(* Logix 5000 project; controller QA_DC vendor 1 type 14 code 164 rev 32.16; software revision 32.04; part 2 of 3 *)
(* tags used below, declared in another part *)
   LN98_1st_Station_Break_Code : DINT;
   LN98_Break_LineWide : BOOL;
   LN98_FROM_DC1_MAIN_MESSAGES : DINT[20];
   LN98_Schedule : UDT_Current_Status;
   LN98_TO_DC1_MAIN_MESSAGE_E : DINT[10];   // WORK CENTER E CONSUME TAG
   LN98_TO_DC1_SUB_MESSAGE_E : DINT[10];   // WORK CENTER E CONSUME TAG
   LN98EES01 : DINT;
   LN98EES02 : DINT;
   LN98EES03 : DINT;
   LN98NEM02 : DINT;
   LN98NEM03 : DINT;
   LN98NEM04 : DINT;
   LN98NEM05 : DINT;
   LN98SEM02 : DINT;
   LN98SEM04 : DINT;
   LN98SEM05 : DINT;
   LN98WES01 : DINT;
   LN98WES02 : DINT;
   LN98WES03 : DINT;
   LN99_1st_Station_Break_Code : DINT;
   LN99_Break_LineWide : BOOL;
   LN99_Current_Shift_Duration_Mins : DINT;
   LN99_Current_Shift_Duration_wBreaks_Mins : DINT;
   LN99_DC_Controlled_Theoretical_Units : BOOL;
   LN99_DT_CODE : DINT;
   LN99_NewDataModelSerial : BOOL;
   LN99_PreviousSerialNumber : STRING;
   LN99_Schedule : UDT_Current_Status;
   LN99_Schedule_Cycle_Timer : TIMER;
   LN99_Schedule_Max_Break_Duration : DINT;
   LN99_Schedule_Max_Break_Timer : TIMER;
   LN99_Schedule_TAKT : REAL;
   LN99_Scheduled_Units_Buffer : DINT;
   LN99_SerialNumber_ONS : BOOL;
   LN99_SerialNumberBuffer : STRING;
   LN99_SerialNumberChange_DelayTimer : TIMER;
   LN99_SerialNumberChange_Timer : TIMER;
   LN99_Shift_Reset_ONS : BOOL;
   LN99_Theoretical_Units_Counter : COUNTER;
   LN99_Theoretical_Units_Counter_ONS : BOOL;
   LN99_TO_DC01_DOWNTIME_CODE : DINT[10];   // DOWNTIME CODE CONSUME TAG
   LN99_TO_DC01_MAIN_MESSAGES : DINT[20];   // KPI CONSUME TAG
   LN99_TO_DC01_MODEL_SERIAL_MESSAGE : STRING[2];
   LN99_TO_DC1_MAIN_MESSAGE_A : DINT[10];   // WORK CENTER A CONSUME TAG
   LN99_TO_DC1_MAIN_MESSAGE_B : DINT[10];   // WORK CENTER B CONSUME TAG
   LN99_TO_DC1_MAIN_MESSAGE_C : DINT[10];   // WORK CENTER C CONSUME TAG
   LN99_Weekly_Schedule : UDT_Weekly_Schedule;
   LN99_WORKCENTER_MAINLINE_A_DT_CODE : DINT;
   LN99_WORKCENTER_MAINLINE_B_DT_CODE : DINT;
   LN99_WORKCENTER_MAINLINE_C_DT_CODE : DINT;
   LN99_WORKCENTER_MAINLINE_D_DT_CODE : DINT;
   LN99_WORKCENTER_MAINLINE_E_DT_CODE : DINT;
   LN99_WORKCENTER_SUBLINE_C_DT_CODE : DINT;
   LN99_WORKCENTER_SUBLINE_E_DT_CODE : DINT;
   LN99NAM01 : DINT;   // WORKSTATION NORTH SIDE WORKCENTER A MAIN LINE STATION 01
   LN99NAM02 : DINT;   // WORKSTATION NORTH SIDE WORKCENTER A MAINLINE STATION 02
   LN99NAM03 : DINT;   // WORKSTATION NORTH SIDE WORKCENTER A MAINLINE STATION 03
   LN99NAM04 : DINT;   // WORKSTATION NORTH SIDE WORKCENTER A MAINLINE STATION 04
   LN99NBM01 : DINT;   // WORK STATION NORTH SIDE WORKCENTER B MAINLINE STATION 01
   LN99NBM02 : DINT;   // WORK STATION NORTH SIDE WORKCENTER B MAINLINE STATION 02
   LN99NBM03 : DINT;   // WORK STATION NORTH SIDE WORKCENTER B MAINLINE STATION 03
   LN99NBM04 : DINT;   // WORK STATION NORTH SIDE WORKCENTER B MAINLINE STATION 4
   LN99NCM01 : DINT;   // WORK STATION NORTH SIDE WORKCENTER C MAINLINE STATION 01
   LN99NCM02 : DINT;   // WORK STATION NORTH SIDE WORKCENTER C MAINLINE STATION 02
   LN99NCM04 : DINT;   // WORK STATION NORTH SIDE WORKCENTER C MAINLINE STATION 04
   LN99NCM05 : DINT;   // WORK STATION NORTH SIDE WORKCENTER C MAINLINE STATION 05
   LN99SAM01 : DINT;   // WORKSTATION SOUTH SIDE WORKCENTER A MAIN LINE STATION 01
   LN99SAM02 : DINT;   // WORKSTATION SOUTH SIDE WORKCENTER A MAINLINE STATION 02
   LN99SAM03 : DINT;   // WORKSTATION SOUTH SIDE WORKCENTER A MAINLINE STATION 03
   LN99SAM04 : DINT;   // WORKSTATION SOUTH SIDE WORKCENTER A MAINLINE STATION 04
   LN99SBM01 : DINT;   // WORK STATION SOUTH SIDE WORKCENTER B MAINLINE STATION 01
   LN99SBM02 : DINT;   // WORK STATION SOUTH SIDE WORKCENTER B MAINLINE STATION 02
   LN99SBM03 : DINT;   // WORK STATION SOUTH SIDE WORKCENTER B MAINLINE STATION 03
   LN99SBM04 : DINT;   // WORK STATION SOUTH SIDE WORKCENTER B MAINLINE STATION 04
   LN99SCM01 : DINT;   // WORK STATION SOUTH SIDE WORKCENTER C MAINLINE STATION 01
   LN99SCM02 : DINT;   // WORK STATION SOUTH SIDE WORKCENTER C MAINLINE STATION 02
   LN99SCM03 : DINT;   // WORK STATION SOUTH SIDE WORKCENTER C MAINLINE STATION 03
   LN99SCM04 : DINT;   // WORK STATION SOUTH SIDE WORKCENTER C MAINLINE STATION 04
   LN99SCM05 : DINT;   // WORK STATION SOUTH SIDE WORKCENTER C MAINLINE STATION 05
(* LN98, continued *)

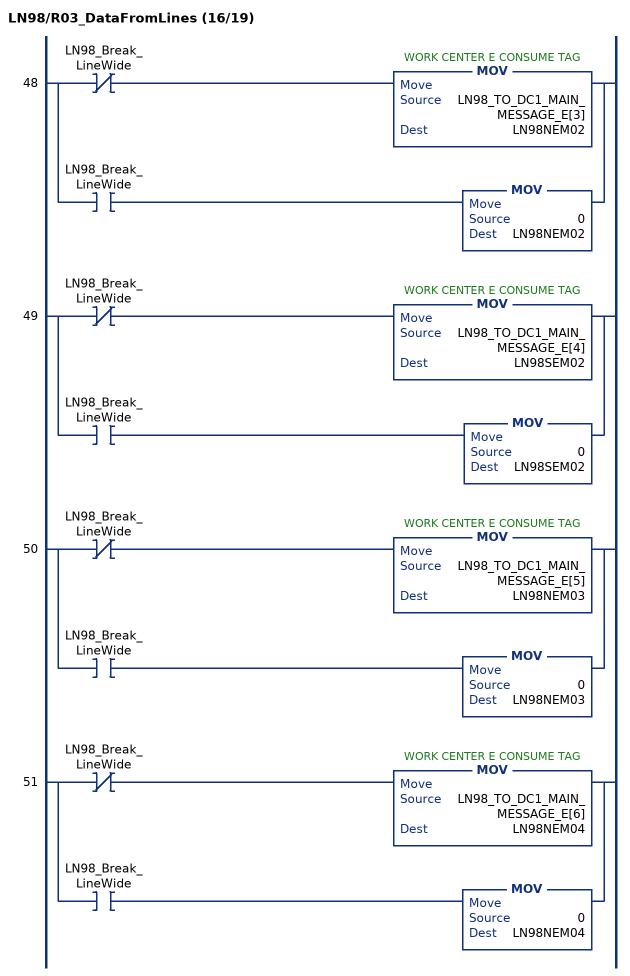
   48: [XIO(LN98_Break_LineWide) MOV(LN98_TO_DC1_MAIN_MESSAGE_E[3],LN98NEM02) ,XIC(LN98_Break_LineWide) MOV(0,LN98NEM02) ];
   49: [XIO(LN98_Break_LineWide) MOV(LN98_TO_DC1_MAIN_MESSAGE_E[4],LN98SEM02) ,XIC(LN98_Break_LineWide) MOV(0,LN98SEM02) ];
   50: [XIO(LN98_Break_LineWide) MOV(LN98_TO_DC1_MAIN_MESSAGE_E[5],LN98NEM03) ,XIC(LN98_Break_LineWide) MOV(0,LN98NEM03) ];
   51: [XIO(LN98_Break_LineWide) MOV(LN98_TO_DC1_MAIN_MESSAGE_E[6],LN98NEM04) ,XIC(LN98_Break_LineWide) MOV(0,LN98NEM04) ];
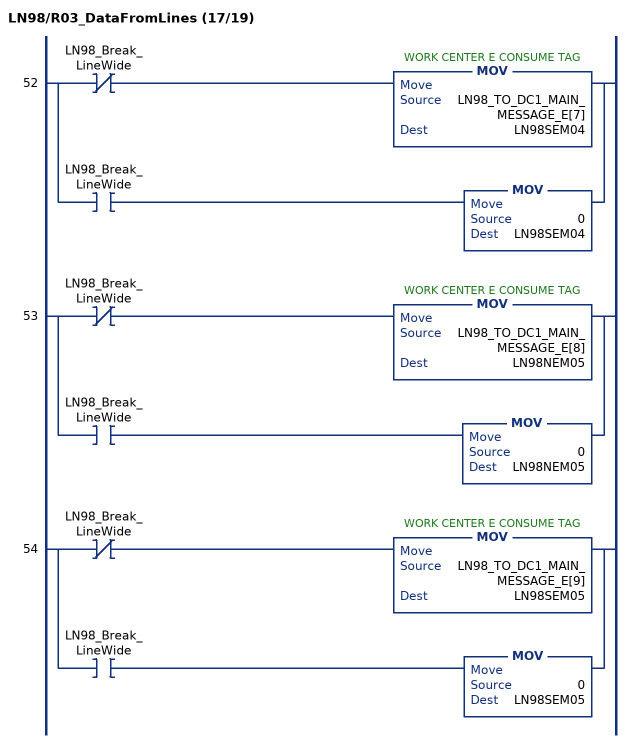
   52: [XIO(LN98_Break_LineWide) MOV(LN98_TO_DC1_MAIN_MESSAGE_E[7],LN98SEM04) ,XIC(LN98_Break_LineWide) MOV(0,LN98SEM04) ];
   53: [XIO(LN98_Break_LineWide) MOV(LN98_TO_DC1_MAIN_MESSAGE_E[8],LN98NEM05) ,XIC(LN98_Break_LineWide) MOV(0,LN98NEM05) ];
   54: [XIO(LN98_Break_LineWide) MOV(LN98_TO_DC1_MAIN_MESSAGE_E[9],LN98SEM05) ,XIC(LN98_Break_LineWide) MOV(0,LN98SEM05) ];
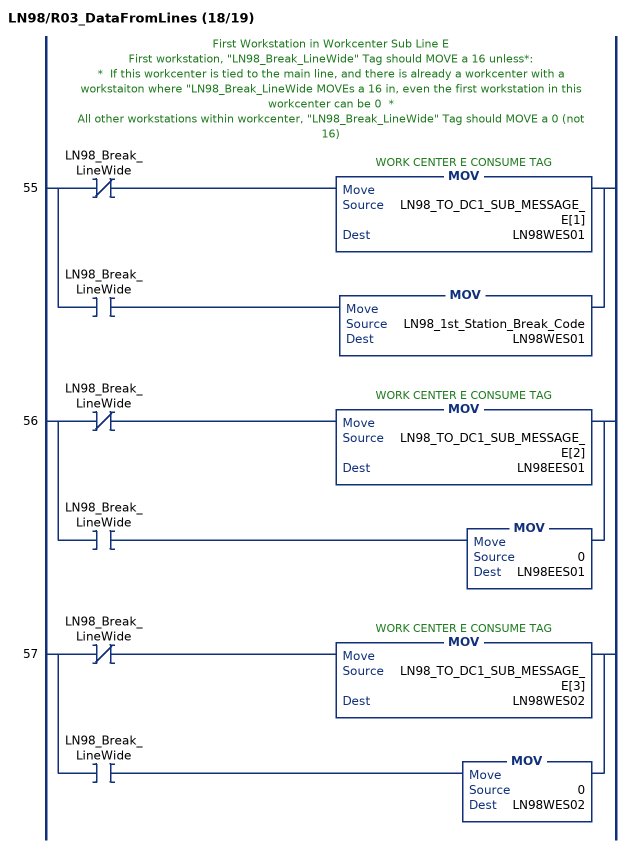
   // First Workstation in Workcenter Sub Line E
   // First workstation, "LN98_Break_LineWide" Tag should MOVE a 16 unless*:
   // *  If this workcenter is tied to the main line, and there is already a workcenter with a workstaiton where "LN98_Break_LineWide MOVEs a 16 in, even the first workstation in this workcenter can be 0  *
   // All other workstations within workcenter, "LN98_Break_LineWide" Tag should MOVE a 0 (not 16)
   55: [XIO(LN98_Break_LineWide) MOV(LN98_TO_DC1_SUB_MESSAGE_E[1],LN98WES01) ,XIC(LN98_Break_LineWide) MOV(LN98_1st_Station_Break_Code,LN98WES01) ];
   56: [XIO(LN98_Break_LineWide) MOV(LN98_TO_DC1_SUB_MESSAGE_E[2],LN98EES01) ,XIC(LN98_Break_LineWide) MOV(0,LN98EES01) ];
   57: [XIO(LN98_Break_LineWide) MOV(LN98_TO_DC1_SUB_MESSAGE_E[3],LN98WES02) ,XIC(LN98_Break_LineWide) MOV(0,LN98WES02) ];
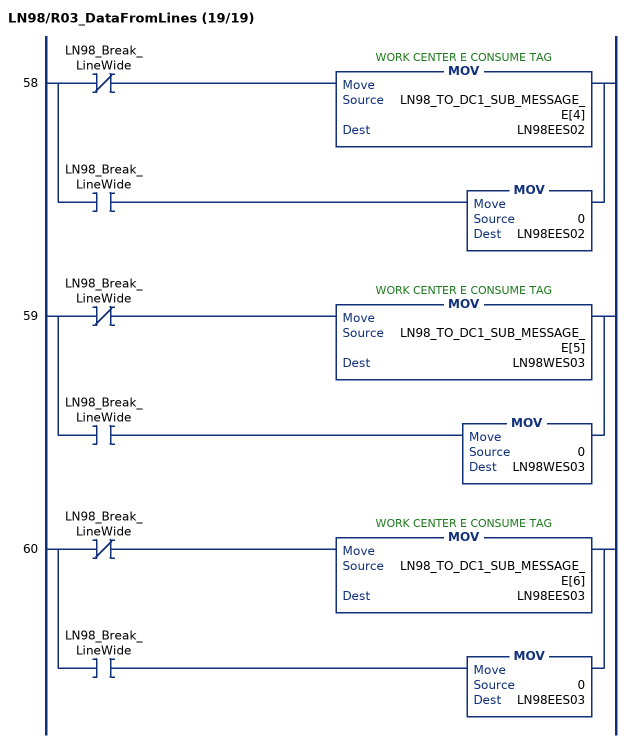
   58: [XIO(LN98_Break_LineWide) MOV(LN98_TO_DC1_SUB_MESSAGE_E[4],LN98EES02) ,XIC(LN98_Break_LineWide) MOV(0,LN98EES02) ];
   59: [XIO(LN98_Break_LineWide) MOV(LN98_TO_DC1_SUB_MESSAGE_E[5],LN98WES03) ,XIC(LN98_Break_LineWide) MOV(0,LN98WES03) ];
   60: [XIO(LN98_Break_LineWide) MOV(LN98_TO_DC1_SUB_MESSAGE_E[6],LN98EES03) ,XIC(LN98_Break_LineWide) MOV(0,LN98EES03) ];
END_ROUTINE

ROUTINE R04_DataToLines   (* ladder *)
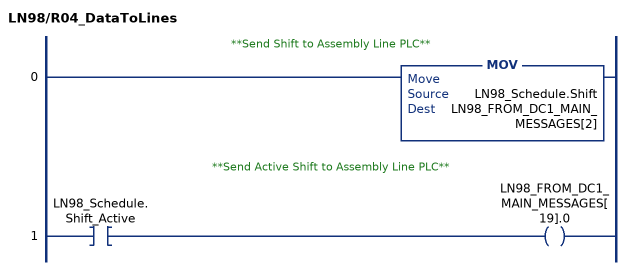
   // **Send Shift to Assembly Line PLC**
   0: MOV(LN98_Schedule.Shift,LN98_FROM_DC1_MAIN_MESSAGES[2]);
   // **Send Active Shift to Assembly Line PLC**
   1: XIC(LN98_Schedule.Shift_Active)OTE(LN98_FROM_DC1_MAIN_MESSAGES[19].0);
END_ROUTINE
END_PROGRAM

PROGRAM LN99   (* main routine MainRoutine *)

ROUTINE MainRoutine   (* ladder *)
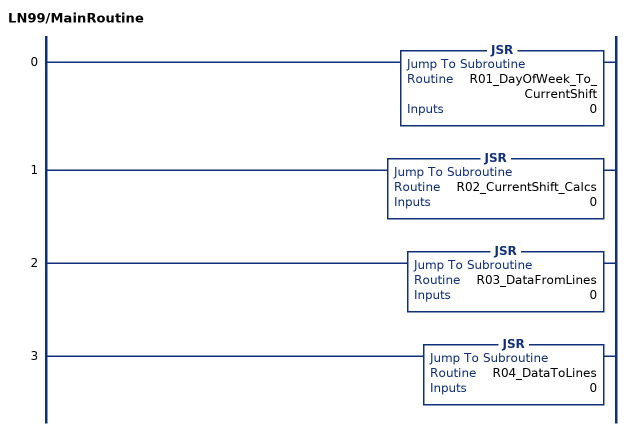
   0: JSR(R01_DayOfWeek_To_CurrentShift,0);
   1: JSR(R02_CurrentShift_Calcs,0);
   2: JSR(R03_DataFromLines,0);
   3: JSR(R04_DataToLines,0);
END_ROUTINE

ROUTINE R01_DayOfWeek_To_CurrentShift   (* ladder *)
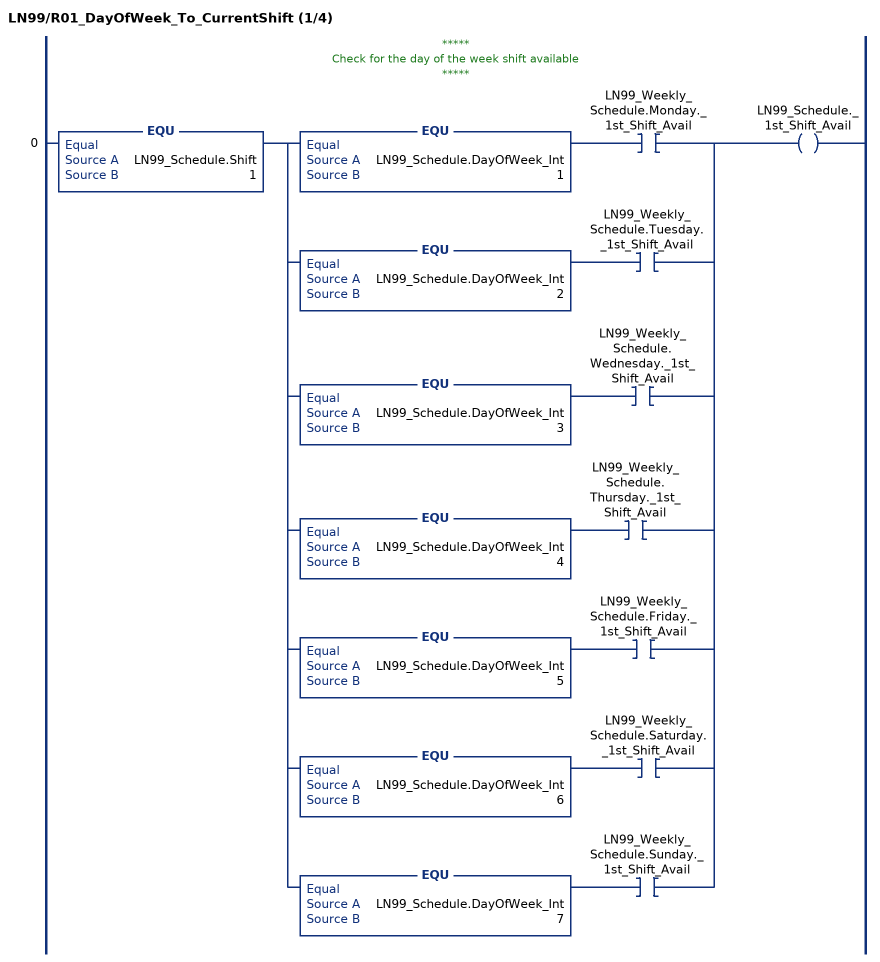
   // *****
   // Check for the day of the week shift available
   // *****
   0: EQU(LN99_Schedule.Shift,1)[EQU(LN99_Schedule.DayOfWeek_Int,1) XIC(LN99_Weekly_Schedule.Monday._1st_Shift_Avail) ,EQU(LN99_Schedule.DayOfWeek_Int,2) XIC(LN99_Weekly_Schedule.Tuesday._1st_Shift_Avail) ,EQU(LN99_Schedule.DayOfWeek_Int,3) XIC(LN99_Weekly_Schedule.Wednesday._1st_Shift_Avail) ,EQU(LN99_Schedule.DayOfWeek_Int,4) XIC(LN99_Weekly_Schedule.Thursday._1st_Shift_Avail) ,EQU(LN99_Schedule.DayOfWeek_Int,5) XIC(LN99_Weekly_Schedule.Friday._1st_Shift_Avail) ,EQU(LN99_Schedule.DayOfWeek_Int,6) XIC(LN99_Weekly_Schedule.Saturday._1st_Shift_Avail) ,EQU(LN99_Schedule.DayOfWeek_Int,7) XIC(LN99_Weekly_Schedule.Sunday._1st_Shift_Avail) ]OTE(LN99_Schedule._1st_Shift_Avail);
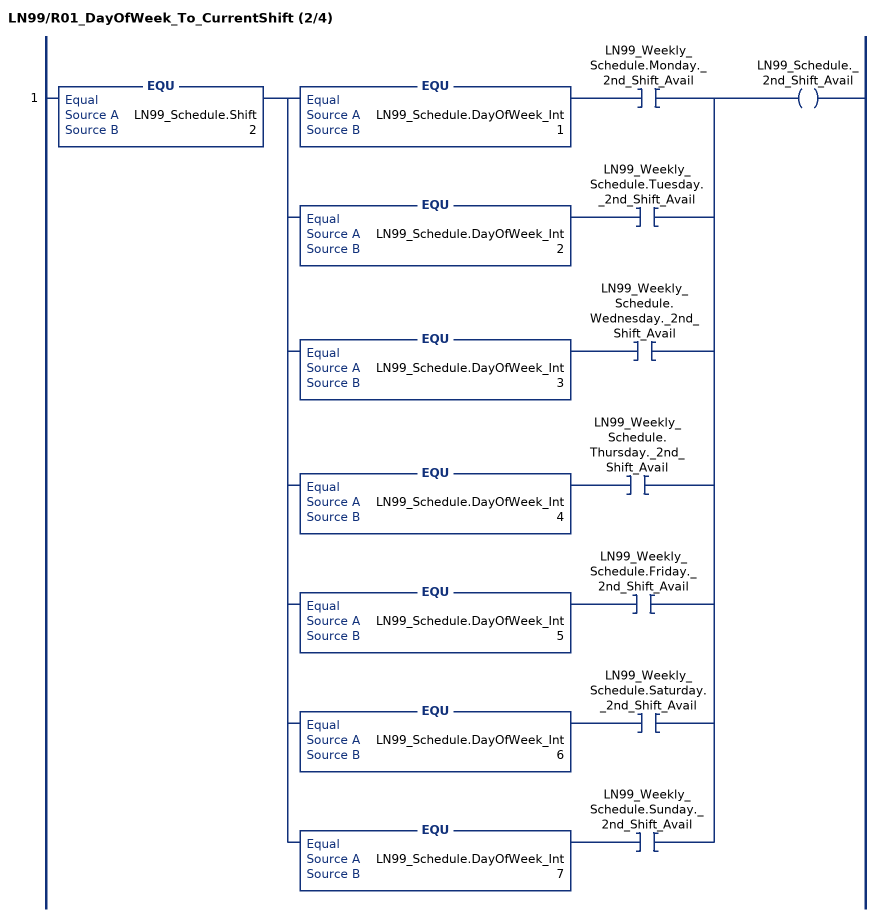
   1: EQU(LN99_Schedule.Shift,2)[EQU(LN99_Schedule.DayOfWeek_Int,1) XIC(LN99_Weekly_Schedule.Monday._2nd_Shift_Avail) ,EQU(LN99_Schedule.DayOfWeek_Int,2) XIC(LN99_Weekly_Schedule.Tuesday._2nd_Shift_Avail) ,EQU(LN99_Schedule.DayOfWeek_Int,3) XIC(LN99_Weekly_Schedule.Wednesday._2nd_Shift_Avail) ,EQU(LN99_Schedule.DayOfWeek_Int,4) XIC(LN99_Weekly_Schedule.Thursday._2nd_Shift_Avail) ,EQU(LN99_Schedule.DayOfWeek_Int,5) XIC(LN99_Weekly_Schedule.Friday._2nd_Shift_Avail) ,EQU(LN99_Schedule.DayOfWeek_Int,6) XIC(LN99_Weekly_Schedule.Saturday._2nd_Shift_Avail) ,EQU(LN99_Schedule.DayOfWeek_Int,7) XIC(LN99_Weekly_Schedule.Sunday._2nd_Shift_Avail) ]OTE(LN99_Schedule._2nd_Shift_Avail);
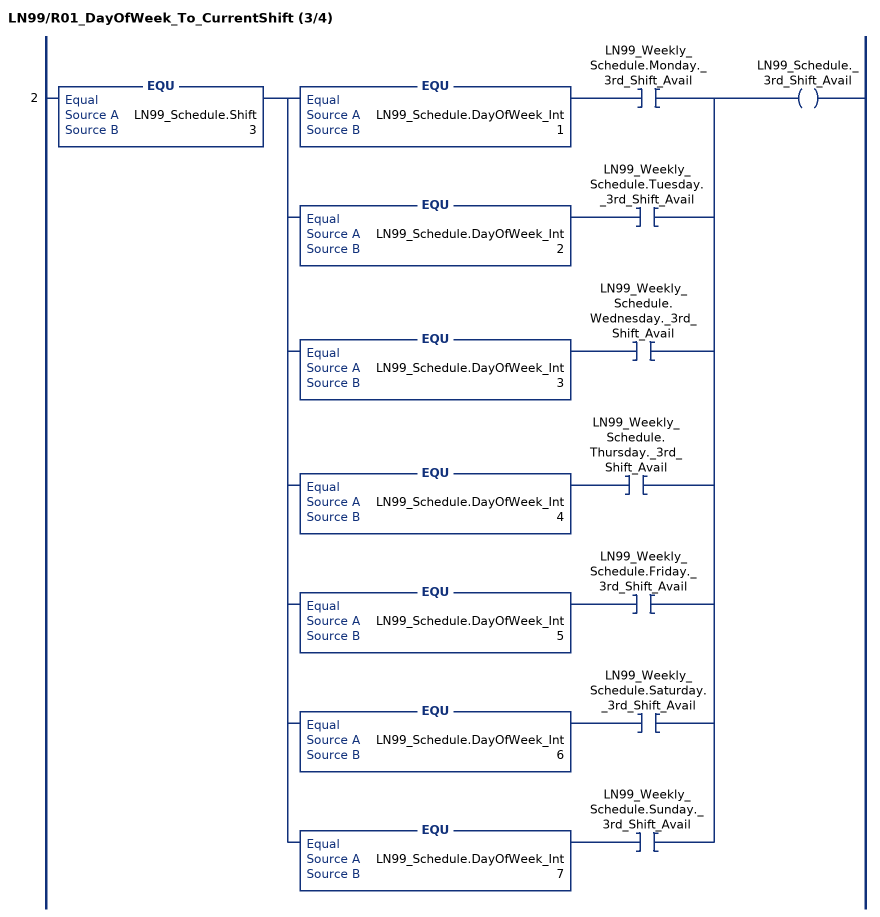
   2: EQU(LN99_Schedule.Shift,3)[EQU(LN99_Schedule.DayOfWeek_Int,1) XIC(LN99_Weekly_Schedule.Monday._3rd_Shift_Avail) ,EQU(LN99_Schedule.DayOfWeek_Int,2) XIC(LN99_Weekly_Schedule.Tuesday._3rd_Shift_Avail) ,EQU(LN99_Schedule.DayOfWeek_Int,3) XIC(LN99_Weekly_Schedule.Wednesday._3rd_Shift_Avail) ,EQU(LN99_Schedule.DayOfWeek_Int,4) XIC(LN99_Weekly_Schedule.Thursday._3rd_Shift_Avail) ,EQU(LN99_Schedule.DayOfWeek_Int,5) XIC(LN99_Weekly_Schedule.Friday._3rd_Shift_Avail) ,EQU(LN99_Schedule.DayOfWeek_Int,6) XIC(LN99_Weekly_Schedule.Saturday._3rd_Shift_Avail) ,EQU(LN99_Schedule.DayOfWeek_Int,7) XIC(LN99_Weekly_Schedule.Sunday._3rd_Shift_Avail) ]OTE(LN99_Schedule._3rd_Shift_Avail);
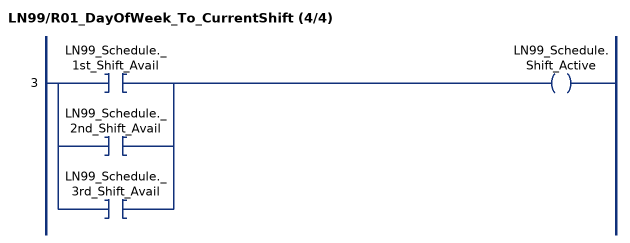
   3: [XIC(LN99_Schedule._1st_Shift_Avail) ,XIC(LN99_Schedule._2nd_Shift_Avail) ,XIC(LN99_Schedule._3rd_Shift_Avail) ]OTE(LN99_Schedule.Shift_Active);
END_ROUTINE

ROUTINE R02_CurrentShift_Calcs   (* ladder *)
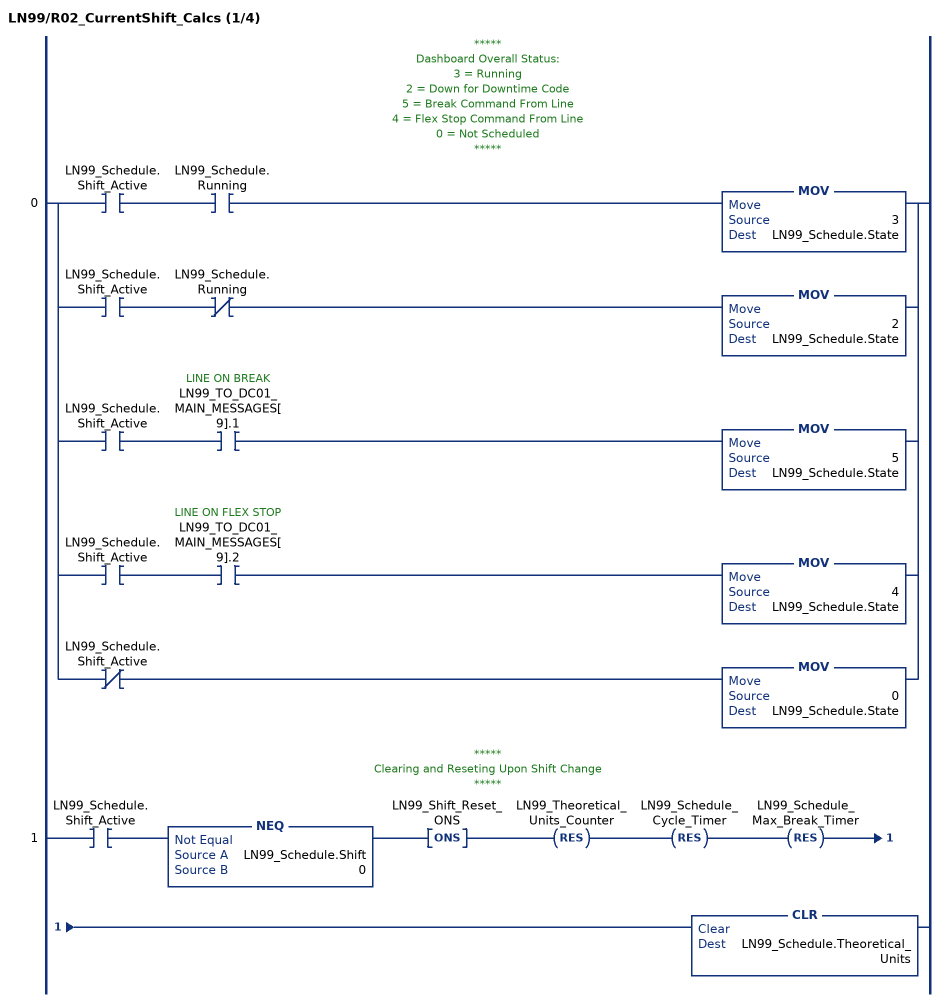
   // *****
   // Dashboard Overall Status:
   // 3 = Running
   // 2 = Down for Downtime Code
   // 5 = Break Command From Line
   // 4 = Flex Stop Command From Line
   // 0 = Not Scheduled
   // *****
   0: [XIC(LN99_Schedule.Shift_Active) XIC(LN99_Schedule.Running) MOV(3,LN99_Schedule.State) ,XIC(LN99_Schedule.Shift_Active) XIO(LN99_Schedule.Running) MOV(2,LN99_Schedule.State) ,XIC(LN99_Schedule.Shift_Active) XIC(LN99_TO_DC01_MAIN_MESSAGES[9].1) MOV(5,LN99_Schedule.State) ,XIC(LN99_Schedule.Shift_Active) XIC(LN99_TO_DC01_MAIN_MESSAGES[9].2) MOV(4,LN99_Schedule.State) ,XIO(LN99_Schedule.Shift_Active) MOV(0,LN99_Schedule.State) ];
   // *****
   // Clearing and Reseting Upon Shift Change
   // *****
   1: XIC(LN99_Schedule.Shift_Active)NEQ(LN99_Schedule.Shift,0)ONS(LN99_Shift_Reset_ONS)RES(LN99_Theoretical_Units_Counter)RES(LN99_Schedule_Cycle_Timer)RES(LN99_Schedule_Max_Break_Timer)CLR(LN99_Schedule.Theoretical_Units);
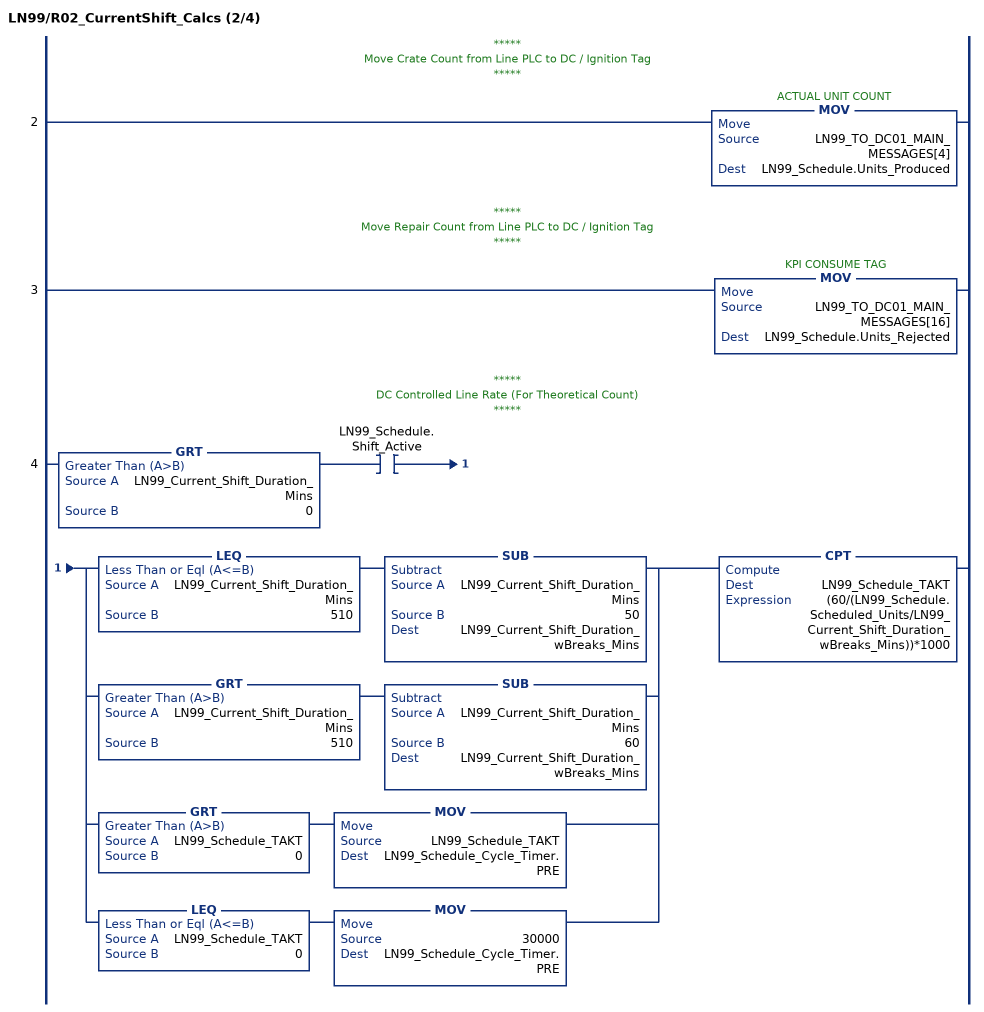
   // *****
   // Move Crate Count from Line PLC to DC / Ignition Tag
   // *****
   2: MOV(LN99_TO_DC01_MAIN_MESSAGES[4],LN99_Schedule.Units_Produced);
   // *****
   // Move Repair Count from Line PLC to DC / Ignition Tag
   // *****
   3: MOV(LN99_TO_DC01_MAIN_MESSAGES[16],LN99_Schedule.Units_Rejected);
   // *****
   // DC Controlled Line Rate (For Theoretical Count)
   // *****
   4: GRT(LN99_Current_Shift_Duration_Mins,0)XIC(LN99_Schedule.Shift_Active)[LEQ(LN99_Current_Shift_Duration_Mins,510) SUB(LN99_Current_Shift_Duration_Mins,50,LN99_Current_Shift_Duration_wBreaks_Mins) ,GRT(LN99_Current_Shift_Duration_Mins,510) SUB(LN99_Current_Shift_Duration_Mins,60,LN99_Current_Shift_Duration_wBreaks_Mins) ,GRT(LN99_Schedule_TAKT,0) MOV(LN99_Schedule_TAKT,LN99_Schedule_Cycle_Timer.PRE) ,LEQ(LN99_Schedule_TAKT,0) MOV(30000,LN99_Schedule_Cycle_Timer.PRE) ]CPT(LN99_Schedule_TAKT,(60/(LN99_Schedule.Scheduled_Units/LN99_Current_Shift_Duration_wBreaks_Mins))*1000);
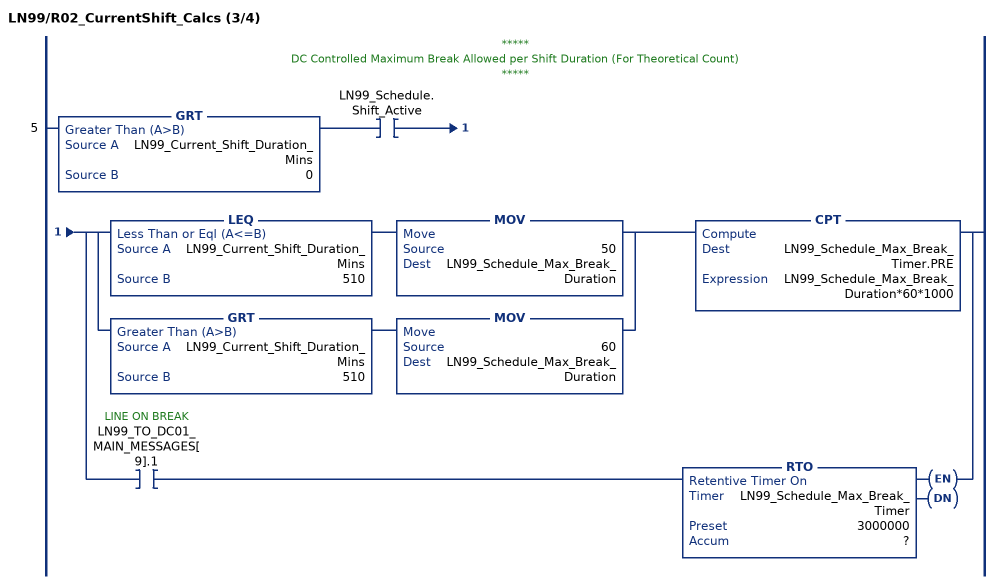
   // *****
   // DC Controlled Maximum Break Allowed per Shift Duration (For Theoretical Count)
   // *****
   5: GRT(LN99_Current_Shift_Duration_Mins,0)XIC(LN99_Schedule.Shift_Active)[[LEQ(LN99_Current_Shift_Duration_Mins,510) MOV(50,LN99_Schedule_Max_Break_Duration) ,GRT(LN99_Current_Shift_Duration_Mins,510) MOV(60,LN99_Schedule_Max_Break_Duration) ] CPT(LN99_Schedule_Max_Break_Timer.PRE,LN99_Schedule_Max_Break_Duration*60*1000) ,XIC(LN99_TO_DC01_MAIN_MESSAGES[9].1) RTO(LN99_Schedule_Max_Break_Timer,?,?) ];
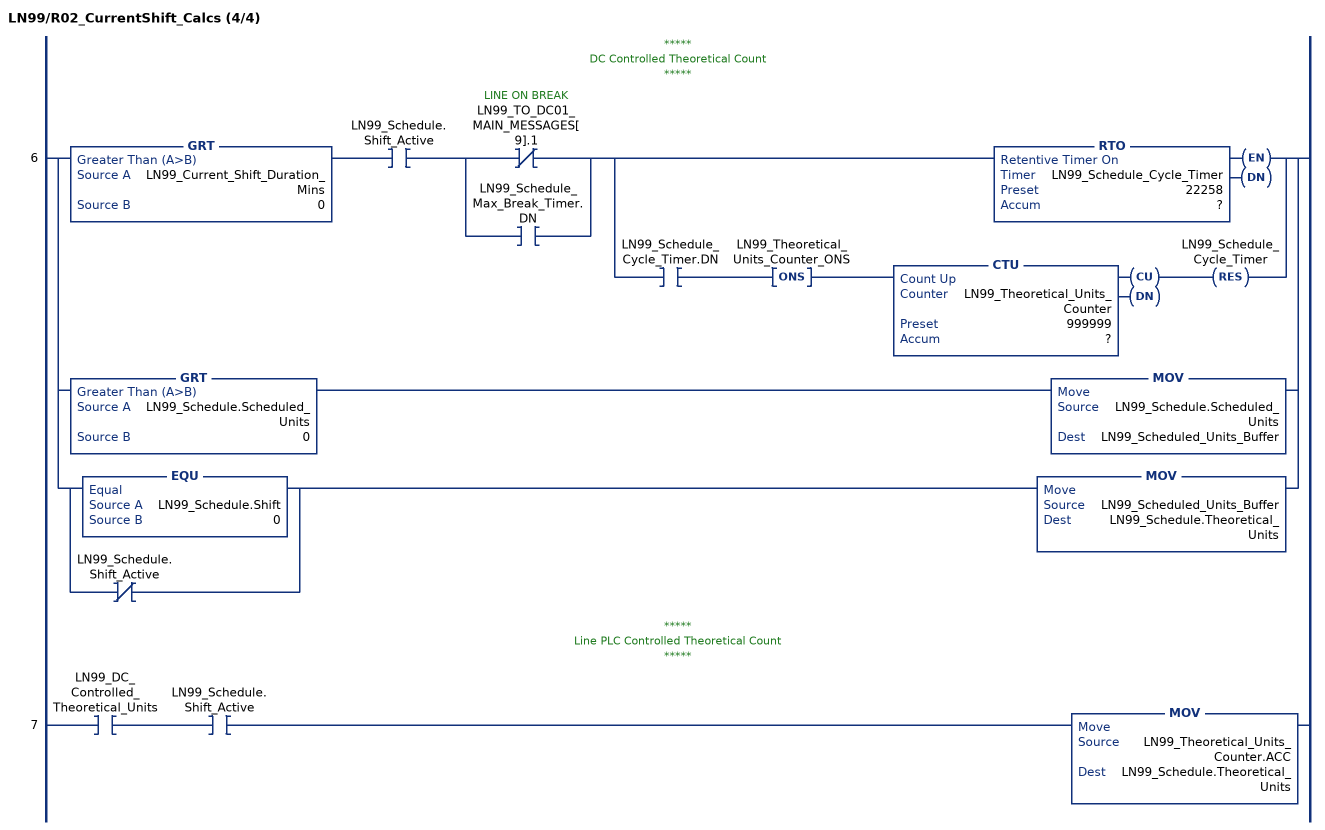
   // *****
   // DC Controlled Theoretical Count
   // *****
   6: [GRT(LN99_Current_Shift_Duration_Mins,0) XIC(LN99_Schedule.Shift_Active) [XIO(LN99_TO_DC01_MAIN_MESSAGES[9].1) ,XIC(LN99_Schedule_Max_Break_Timer.DN) ] [RTO(LN99_Schedule_Cycle_Timer,?,?) ,XIC(LN99_Schedule_Cycle_Timer.DN) ONS(LN99_Theoretical_Units_Counter_ONS) CTU(LN99_Theoretical_Units_Counter,?,?) RES(LN99_Schedule_Cycle_Timer) ] ,GRT(LN99_Schedule.Scheduled_Units,0) MOV(LN99_Schedule.Scheduled_Units,LN99_Scheduled_Units_Buffer) ,[EQU(LN99_Schedule.Shift,0) ,XIO(LN99_Schedule.Shift_Active) ] MOV(LN99_Scheduled_Units_Buffer,LN99_Schedule.Theoretical_Units) ];
   // *****
   // Line PLC Controlled Theoretical Count
   // *****
   7: XIC(LN99_DC_Controlled_Theoretical_Units)XIC(LN99_Schedule.Shift_Active)MOV(LN99_Theoretical_Units_Counter.ACC,LN99_Schedule.Theoretical_Units);
END_ROUTINE

ROUTINE R03_DataFromLines   (* ladder *)
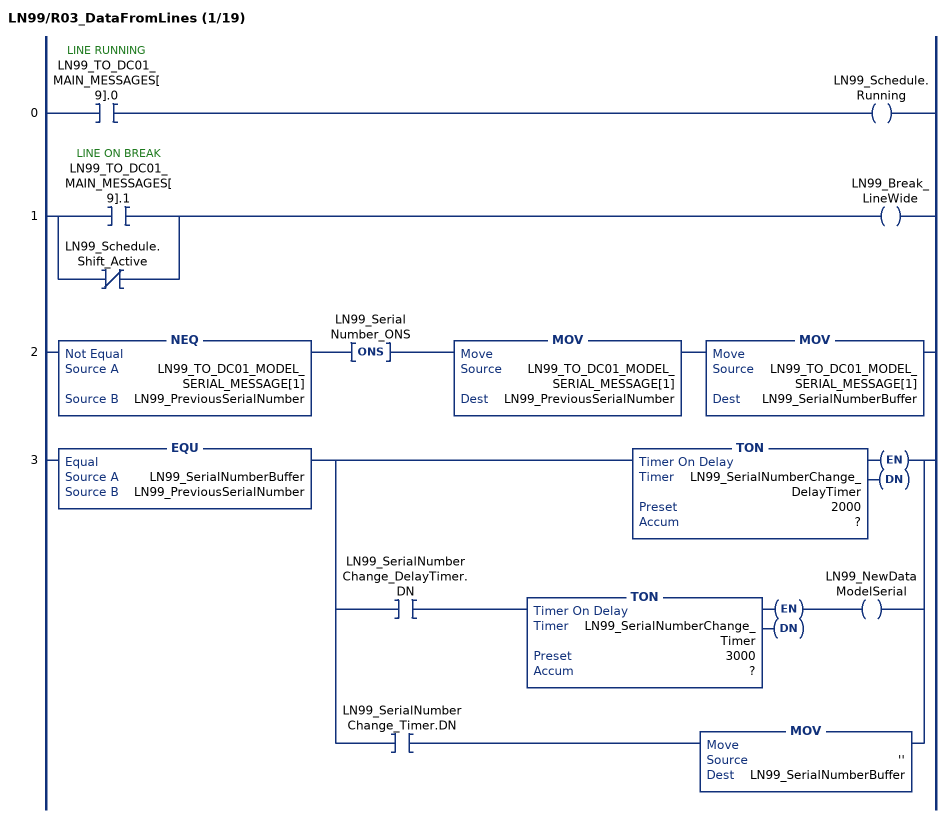
   0: XIC(LN99_TO_DC01_MAIN_MESSAGES[9].0)OTE(LN99_Schedule.Running);
   1: [XIC(LN99_TO_DC01_MAIN_MESSAGES[9].1) ,XIO(LN99_Schedule.Shift_Active) ]OTE(LN99_Break_LineWide);
   2: NEQ(LN99_TO_DC01_MODEL_SERIAL_MESSAGE[1],LN99_PreviousSerialNumber)ONS(LN99_SerialNumber_ONS)MOV(LN99_TO_DC01_MODEL_SERIAL_MESSAGE[1],LN99_PreviousSerialNumber)MOV(LN99_TO_DC01_MODEL_SERIAL_MESSAGE[1],LN99_SerialNumberBuffer);
   3: EQU(LN99_SerialNumberBuffer,LN99_PreviousSerialNumber)[TON(LN99_SerialNumberChange_DelayTimer,?,?) ,XIC(LN99_SerialNumberChange_DelayTimer.DN) TON(LN99_SerialNumberChange_Timer,?,?) OTE(LN99_NewDataModelSerial) ,XIC(LN99_SerialNumberChange_Timer.DN) MOV('',LN99_SerialNumberBuffer) ];
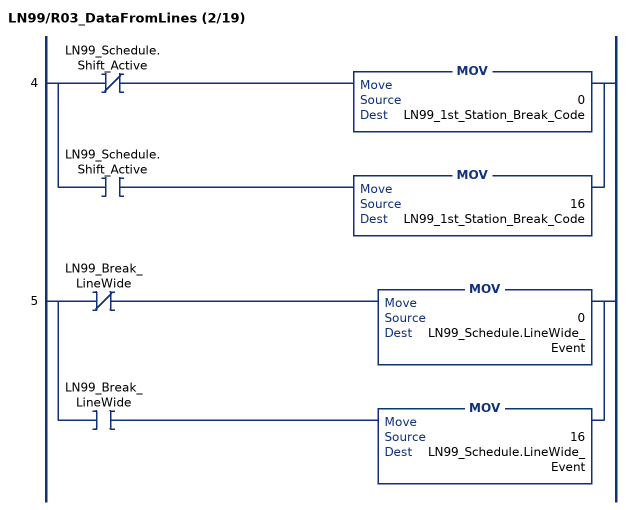
   4: [XIO(LN99_Schedule.Shift_Active) MOV(0,LN99_1st_Station_Break_Code) ,XIC(LN99_Schedule.Shift_Active) MOV(16,LN99_1st_Station_Break_Code) ];
   5: [XIO(LN99_Break_LineWide) MOV(0,LN99_Schedule.LineWide_Event) ,XIC(LN99_Break_LineWide) MOV(16,LN99_Schedule.LineWide_Event) ];
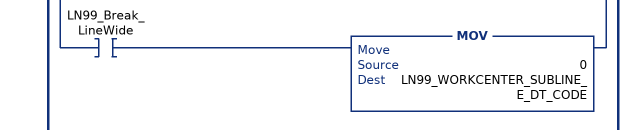
   // MNT Faults
   // If an MNT workcenter is tied to the main line or subline where there is already a workcenter with a workstaiton where "LN99_Break_LineWide (when high) MOVEs a 16 in, then that MNT can MOVE a 0 in when "LN99_Break_LineWide" goes high
   // If it is an independent MNT (not tied to a workcenter), "LN99_Break_LineWide" Tag should MOVE a 16 when "LN99_Break_LineWide" goes high
   6: [XIO(LN99_Break_LineWide) MOV(LN99_TO_DC01_DOWNTIME_CODE[0],LN99_DT_CODE) ,XIC(LN99_Break_LineWide) MOV(0,LN99_DT_CODE) ,XIO(LN99_Break_LineWide) MOV(LN99_TO_DC01_DOWNTIME_CODE[1],LN99_WORKCENTER_MAINLINE_A_DT_CODE) ,XIC(LN99_Break_LineWide) MOV(0,LN99_WORKCENTER_MAINLINE_A_DT_CODE) ,XIO(LN99_Break_LineWide) MOV(LN99_TO_DC01_DOWNTIME_CODE[2],LN99_WORKCENTER_MAINLINE_B_DT_CODE) ,XIC(LN99_Break_LineWide) MOV(0,LN99_WORKCENTER_MAINLINE_B_DT_CODE) ,XIO(LN99_Break_LineWide) MOV(LN99_TO_DC01_DOWNTIME_CODE[3],LN99_WORKCENTER_MAINLINE_C_DT_CODE) ,XIC(LN99_Break_LineWide) MOV(0,LN99_WORKCENTER_MAINLINE_C_DT_CODE) ,XIO(LN99_Break_LineWide) MOV(LN99_TO_DC01_DOWNTIME_CODE[4],LN99_WORKCENTER_MAINLINE_D_DT_CODE) ,XIC(LN99_Break_LineWide) MOV(0,LN99_WORKCENTER_MAINLINE_D_DT_CODE) ,XIO(LN99_Break_LineWide) MOV(LN99_TO_DC01_DOWNTIME_CODE[5],LN99_WORKCENTER_MAINLINE_E_DT_CODE) ,XIC(LN99_Break_LineWide) MOV(0,LN99_WORKCENTER_MAINLINE_E_DT_CODE) ,XIO(LN99_Break_LineWide) MOV(LN99_TO_DC01_DOWNTIME_CODE[6],LN99_WORKCENTER_SUBLINE_C_DT_CODE) ,XIC(LN99_Break_LineWide) MOV(0,LN99_WORKCENTER_SUBLINE_C_DT_CODE) ,XIO(LN99_Break_LineWide) MOV(LN99_TO_DC01_DOWNTIME_CODE[7],LN99_WORKCENTER_SUBLINE_E_DT_CODE) ,XIC(LN99_Break_LineWide) MOV(0,LN99_WORKCENTER_SUBLINE_E_DT_CODE) ];
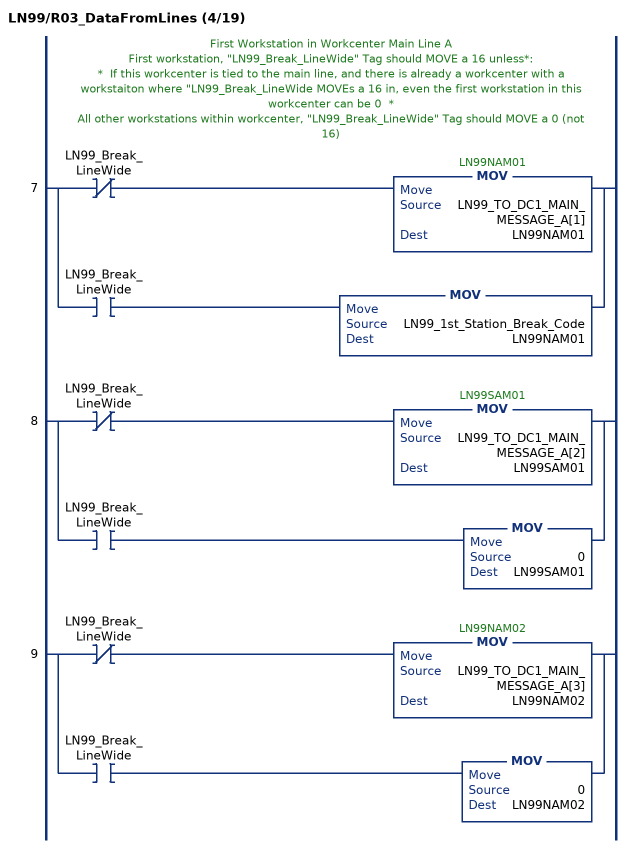
   // First Workstation in Workcenter Main Line A
   // First workstation, "LN99_Break_LineWide" Tag should MOVE a 16 unless*:
   // *  If this workcenter is tied to the main line, and there is already a workcenter with a workstaiton where "LN99_Break_LineWide MOVEs a 16 in, even the first workstation in this workcenter can be 0  *
   // All other workstations within workcenter, "LN99_Break_LineWide" Tag should MOVE a 0 (not 16)
   7: [XIO(LN99_Break_LineWide) MOV(LN99_TO_DC1_MAIN_MESSAGE_A[1],LN99NAM01) ,XIC(LN99_Break_LineWide) MOV(LN99_1st_Station_Break_Code,LN99NAM01) ];
   8: [XIO(LN99_Break_LineWide) MOV(LN99_TO_DC1_MAIN_MESSAGE_A[2],LN99SAM01) ,XIC(LN99_Break_LineWide) MOV(0,LN99SAM01) ];
   9: [XIO(LN99_Break_LineWide) MOV(LN99_TO_DC1_MAIN_MESSAGE_A[3],LN99NAM02) ,XIC(LN99_Break_LineWide) MOV(0,LN99NAM02) ];
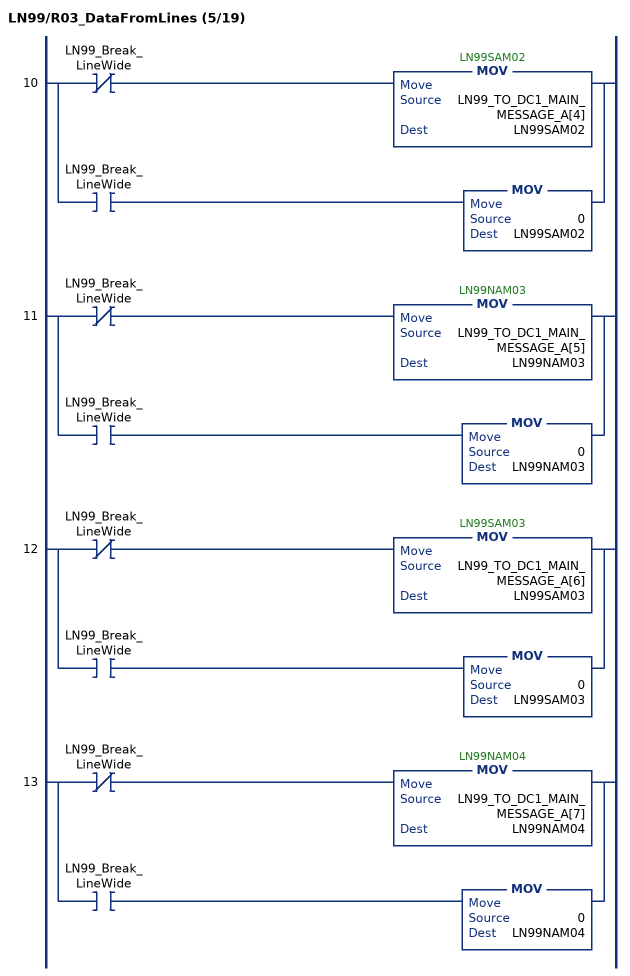
   10: [XIO(LN99_Break_LineWide) MOV(LN99_TO_DC1_MAIN_MESSAGE_A[4],LN99SAM02) ,XIC(LN99_Break_LineWide) MOV(0,LN99SAM02) ];
   11: [XIO(LN99_Break_LineWide) MOV(LN99_TO_DC1_MAIN_MESSAGE_A[5],LN99NAM03) ,XIC(LN99_Break_LineWide) MOV(0,LN99NAM03) ];
   12: [XIO(LN99_Break_LineWide) MOV(LN99_TO_DC1_MAIN_MESSAGE_A[6],LN99SAM03) ,XIC(LN99_Break_LineWide) MOV(0,LN99SAM03) ];
   13: [XIO(LN99_Break_LineWide) MOV(LN99_TO_DC1_MAIN_MESSAGE_A[7],LN99NAM04) ,XIC(LN99_Break_LineWide) MOV(0,LN99NAM04) ];
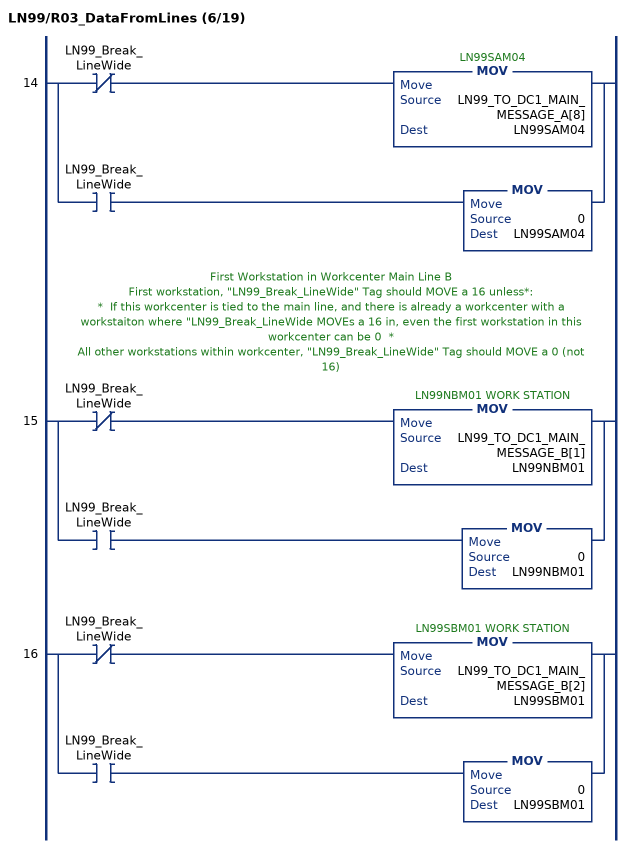
   14: [XIO(LN99_Break_LineWide) MOV(LN99_TO_DC1_MAIN_MESSAGE_A[8],LN99SAM04) ,XIC(LN99_Break_LineWide) MOV(0,LN99SAM04) ];
   // First Workstation in Workcenter Main Line B
   // First workstation, "LN99_Break_LineWide" Tag should MOVE a 16 unless*:
   // *  If this workcenter is tied to the main line, and there is already a workcenter with a workstaiton where "LN99_Break_LineWide MOVEs a 16 in, even the first workstation in this workcenter can be 0  *
   // All other workstations within workcenter, "LN99_Break_LineWide" Tag should MOVE a 0 (not 16)
   15: [XIO(LN99_Break_LineWide) MOV(LN99_TO_DC1_MAIN_MESSAGE_B[1],LN99NBM01) ,XIC(LN99_Break_LineWide) MOV(0,LN99NBM01) ];
   16: [XIO(LN99_Break_LineWide) MOV(LN99_TO_DC1_MAIN_MESSAGE_B[2],LN99SBM01) ,XIC(LN99_Break_LineWide) MOV(0,LN99SBM01) ];
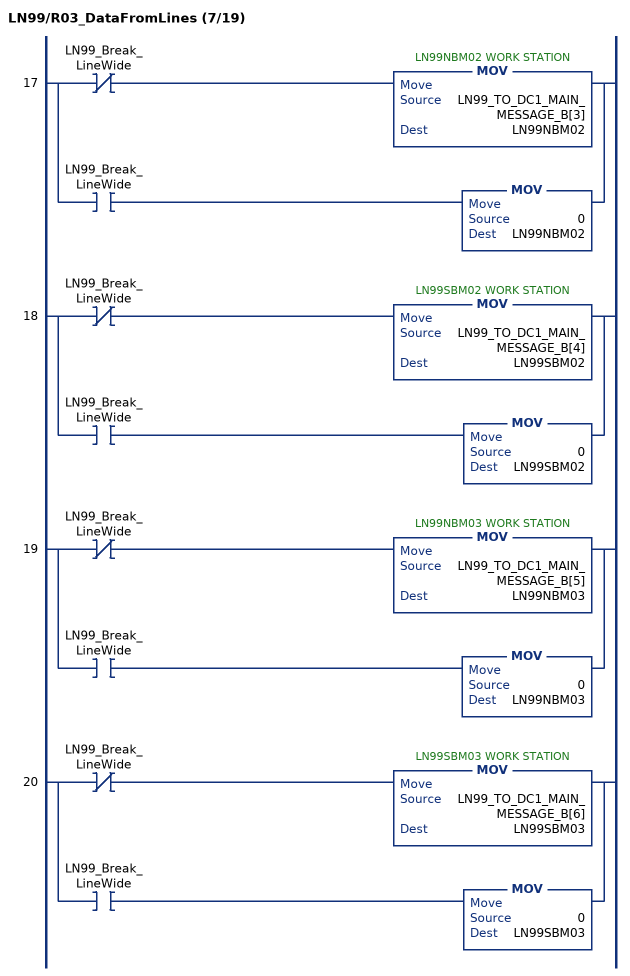
   17: [XIO(LN99_Break_LineWide) MOV(LN99_TO_DC1_MAIN_MESSAGE_B[3],LN99NBM02) ,XIC(LN99_Break_LineWide) MOV(0,LN99NBM02) ];
   18: [XIO(LN99_Break_LineWide) MOV(LN99_TO_DC1_MAIN_MESSAGE_B[4],LN99SBM02) ,XIC(LN99_Break_LineWide) MOV(0,LN99SBM02) ];
   19: [XIO(LN99_Break_LineWide) MOV(LN99_TO_DC1_MAIN_MESSAGE_B[5],LN99NBM03) ,XIC(LN99_Break_LineWide) MOV(0,LN99NBM03) ];
   20: [XIO(LN99_Break_LineWide) MOV(LN99_TO_DC1_MAIN_MESSAGE_B[6],LN99SBM03) ,XIC(LN99_Break_LineWide) MOV(0,LN99SBM03) ];
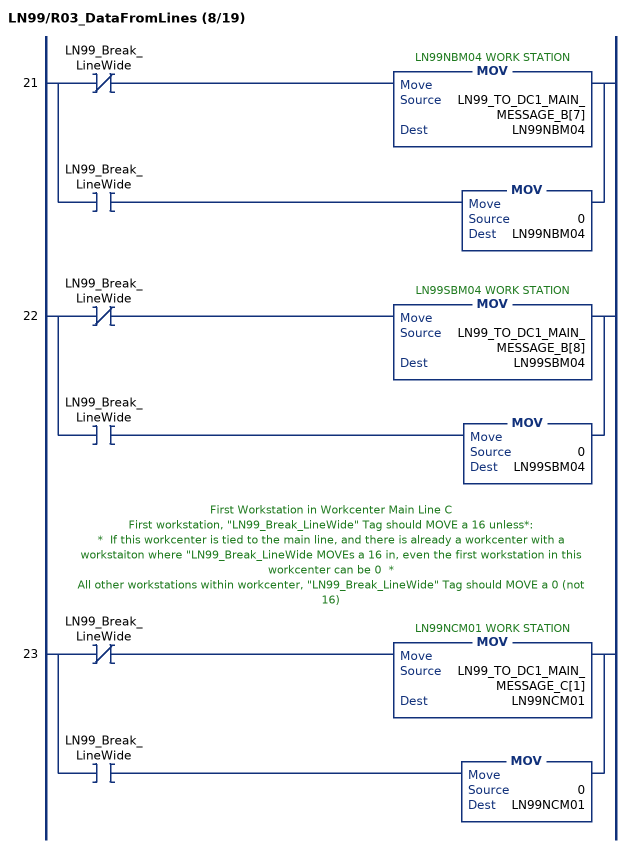
   21: [XIO(LN99_Break_LineWide) MOV(LN99_TO_DC1_MAIN_MESSAGE_B[7],LN99NBM04) ,XIC(LN99_Break_LineWide) MOV(0,LN99NBM04) ];
   22: [XIO(LN99_Break_LineWide) MOV(LN99_TO_DC1_MAIN_MESSAGE_B[8],LN99SBM04) ,XIC(LN99_Break_LineWide) MOV(0,LN99SBM04) ];
   // First Workstation in Workcenter Main Line C
   // First workstation, "LN99_Break_LineWide" Tag should MOVE a 16 unless*:
   // *  If this workcenter is tied to the main line, and there is already a workcenter with a workstaiton where "LN99_Break_LineWide MOVEs a 16 in, even the first workstation in this workcenter can be 0  *
   // All other workstations within workcenter, "LN99_Break_LineWide" Tag should MOVE a 0 (not 16)
   23: [XIO(LN99_Break_LineWide) MOV(LN99_TO_DC1_MAIN_MESSAGE_C[1],LN99NCM01) ,XIC(LN99_Break_LineWide) MOV(0,LN99NCM01) ];
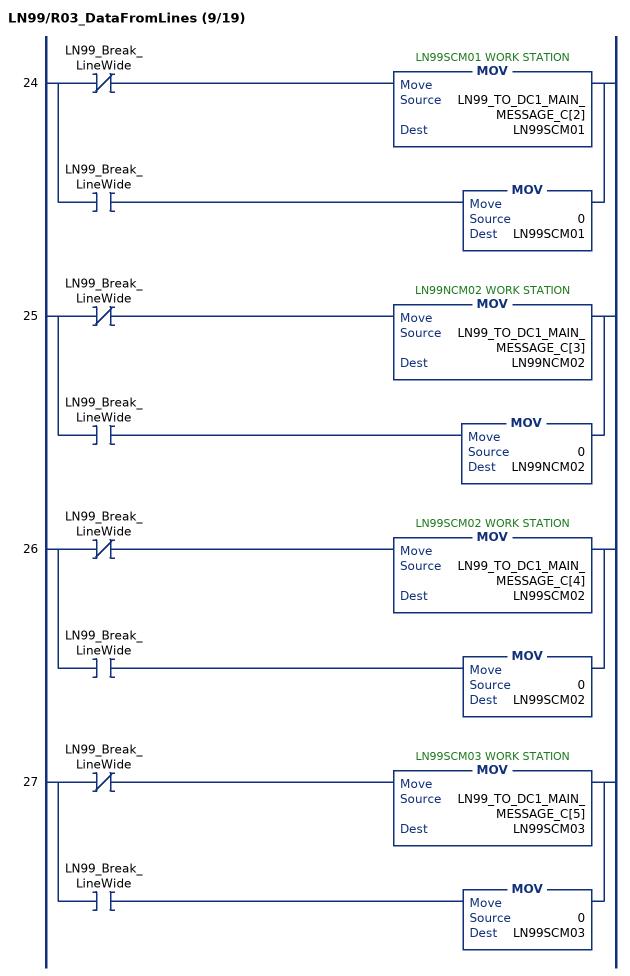
   24: [XIO(LN99_Break_LineWide) MOV(LN99_TO_DC1_MAIN_MESSAGE_C[2],LN99SCM01) ,XIC(LN99_Break_LineWide) MOV(0,LN99SCM01) ];
   25: [XIO(LN99_Break_LineWide) MOV(LN99_TO_DC1_MAIN_MESSAGE_C[3],LN99NCM02) ,XIC(LN99_Break_LineWide) MOV(0,LN99NCM02) ];
   26: [XIO(LN99_Break_LineWide) MOV(LN99_TO_DC1_MAIN_MESSAGE_C[4],LN99SCM02) ,XIC(LN99_Break_LineWide) MOV(0,LN99SCM02) ];
   27: [XIO(LN99_Break_LineWide) MOV(LN99_TO_DC1_MAIN_MESSAGE_C[5],LN99SCM03) ,XIC(LN99_Break_LineWide) MOV(0,LN99SCM03) ];
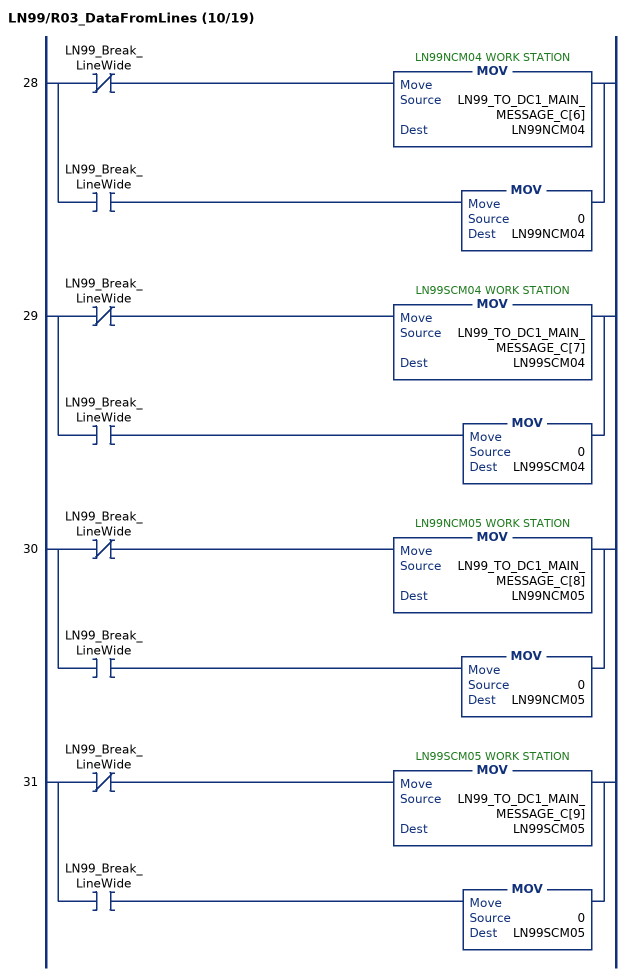
   28: [XIO(LN99_Break_LineWide) MOV(LN99_TO_DC1_MAIN_MESSAGE_C[6],LN99NCM04) ,XIC(LN99_Break_LineWide) MOV(0,LN99NCM04) ];
   29: [XIO(LN99_Break_LineWide) MOV(LN99_TO_DC1_MAIN_MESSAGE_C[7],LN99SCM04) ,XIC(LN99_Break_LineWide) MOV(0,LN99SCM04) ];
   30: [XIO(LN99_Break_LineWide) MOV(LN99_TO_DC1_MAIN_MESSAGE_C[8],LN99NCM05) ,XIC(LN99_Break_LineWide) MOV(0,LN99NCM05) ];
   31: [XIO(LN99_Break_LineWide) MOV(LN99_TO_DC1_MAIN_MESSAGE_C[9],LN99SCM05) ,XIC(LN99_Break_LineWide) MOV(0,LN99SCM05) ];
